{attribute 'qualified_only'}
{attribute 'strict'}
TYPE MC_SYNC_MODE :
(
	enum_member := 0
);
END_TYPE

(* stored: Version 1.1.0.1, ProductVersion 3.1.4024.12
   DUT MC_SYNC_MODE: Id {7a1662ea-6f52-49b3-ad81-2e7f6b6967aa} *)
